Universal Robots PolyScope program: jog.urp

ProgramRoot directory=/programs/usbdisk/JOG; kinematics=(a=[0, -0.425, -0.39225, 0, 0, 0], d=[0.08916, 0, 0, 0.10915, 0.09465, 0.0823], alpha=[1.5708, 0, 0, 1.5708, -1.5708, 0], deltaTheta=[0, 0, 0, 0, 0, 0], status=notInitialized); lastSavedInVersion=(project__name=Polyscope, major__version=3, minor__version=1, svn__revision=17336, build__date=Mar 26 2015, 11:23:02); name=jog; programVersion=(project__name=Polyscope, major__version=3, minor__version=1, svn__revision=17195, build__date=Mar 11 2015, 13:02:28); robotEnvironmentFileName=default; serialNumberRobot=2014350123
  BeforeStart description=COMMAND_SEQUENCE_BEFORE_PROGRAM_START; name=BeforeStart
    Assignment assignmentOperatorMessage=the way of moving; operatorValueType=INTEGER; valueSource=OPERATOR
    Assignment expr=get_actual_tcp_pose(); operatorValueType=INTEGER; valueSource=EXPRESSION
    If expr=ExpressionVariableNode≟1; type=IF_NODE
      Assignment expr=pose_add(p[0,0.1,0,0,0,0],ExpressionVariableNode); operatorValueType=INTEGER; valueSource=EXPRESSION
    If expr=ExpressionVariableNode≟2; type=ELSEIF_NODE
      Assignment expr=pose_add(p[0,0,0,0,1,0],ExpressionVariableNode); operatorValueType=INTEGER; valueSource=EXPRESSION
    If expr=ExpressionVariableNode≟3; type=ELSEIF_NODE
      Assignment expr=pose_trans(ExpressionVariableNode,p[0,0.1,0,0,0,0]); operatorValueType=INTEGER; valueSource=EXPRESSION
    If expr=ExpressionVariableNode≟4; type=ELSEIF_NODE
      Assignment expr=pose_trans(ExpressionVariableNode,p[0,0,0,0,1,0]); operatorValueType=INTEGER; valueSource=EXPRESSION
    If type=ELSE_NODE
      Halt 
  MainProgram cartesianAcceleration=1.2; cartesianSpeed=0.25; jointAcceleration=1.3962634015954636; jointSpeed=1.0471975511965976; sharedProcessMoveBlendRadius=0.025; motionType=JOINT_SPACE
    Move cartesianAcceleration=1.2; cartesianSpeed=0.25; jointAcceleration=1.3962634015954636; jointSpeed=1.0471975511965976; sharedProcessMoveBlendRadius=0.025; motionType=CARTESIAN_SPACE
      Waypoint blendRadius=0.05; cartesianAcceleration=1.2; cartesianSpeed=0.25; jointAcceleration=1.3962634015954636; jointSpeed=1.0471975511965976; nextMotionTime=2.0; stoppoint=true; useSharedBlendParameter=true; useSharedParameters=true; positionType=VARIABLE_POSITION; name=Waypoint
      Waypoint blendRadius=0.05; cartesianAcceleration=1.2; cartesianSpeed=0.25; jointAcceleration=1.3962634015954636; jointSpeed=1.0471975511965976; nextMotionTime=2.0; stoppoint=true; useSharedBlendParameter=true; useSharedParameters=true; positionType=VARIABLE_POSITION; name=Waypoint
